FUNCTION_BLOCK FB_Ambient
VAR_INPUT
END_VAR
VAR_OUTPUT
	{attribute 'OPC.UA.DA' := '1'}
	localState : ST_AmbientState;
END_VAR
VAR
END_VAR

//add ambient temperature rain etc. from weather station
(*
localState.fOutsideTemperature := Umwelt.Temp_Aussen_WS;
localState.bRain := Umwelt.Regen;
localState.fHallTemperature := Umwelt.Temp_Halle_Sektor1;
*)

END_FUNCTION_BLOCK

(* stored: Version 1.1.0.1, ProductVersion 3.1.4024.10
   POU FB_Ambient: Id {e5737b3d-b420-44a4-9ae1-301270e5edfa}, SpecialFunc None *)
